# EPICS substitutions: db/Beckhoff_9XXX/ecmcEL9576.substitutions
file ecmcEcSlave.template
{
  pattern {}
          {}
}

file ecmcEL9576.template
{
  pattern {}
          {}
}
